TYPE AdasData_In :

UNION
	asBin: ARRAY[0..(((gVarL.gVar_NumberOfAdasTracks * 2) + 4) - 1)] OF WORD;
	asData: AdasStreamData;
END_UNION

END_TYPE

(* stored: Version 1.1.0.1, ProductVersion 3.1.4022.16
   DUT AdasData_In: Id {59e71d81-6390-44b3-b35b-db46e3817ee3} *)
